FUNCTION_BLOCK findNext (* Tamplate for a simple Basic Function Block Type *)
  (* Standard: 61499-2 *)
  (* Version 0.0, 2018-01-05, 4DIAC-IDE, 4DIAC-Consortium *)
  (* Version 1.0, 2016-05-26, AZ, fortiss GmbH *)
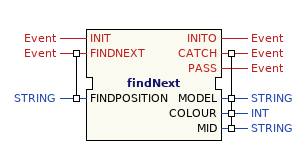
  EVENT_INPUT
    INIT; (* Initialization Request *)
    FINDNEXT WITH FINDPOSITION; (* Normal Execution Request *)
  END_EVENT
  EVENT_OUTPUT
    INITO; (* Initialization Confirm *)
    CATCH WITH MODEL, MID, COLOUR;
    PASS;
  END_EVENT
  VAR_INPUT
    FINDPOSITION : STRING;
  END_VAR
  VAR_OUTPUT
    MODEL : STRING;
    COLOUR : INT;
    MID : STRING;
  END_VAR
  VAR
    catchOrPass : STRING := ''; (* Internal Variable *)
  END_VAR
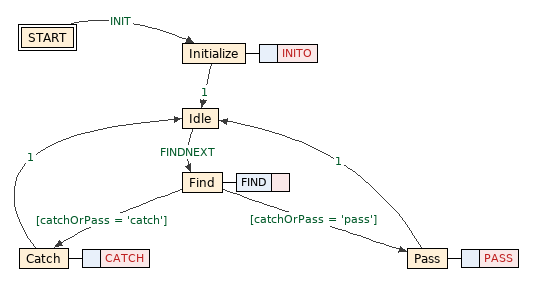
  EC_STATES
    START; (* Initial State *)
    Initialize : -> INITO; (* Initialization *)
    Find : FIND;
    Catch : -> CATCH;
    Pass : -> PASS;
    Idle;
  END_STATES
  EC_TRANSITIONS
    START TO Initialize := INIT;
    Find TO Pass := [catchOrPass = 'pass'];
    Find TO Catch := [catchOrPass = 'catch'];
    Idle TO Find := FINDNEXT;
    Initialize TO Idle := 1;
    Catch TO Idle := 1;
    Pass TO Idle := 1;
  END_TRANSITIONS
  ALGORITHM FIND IN ST: (* new algorithm *)

  END_ALGORITHM
END_FUNCTION_BLOCK
